(* Logix 5000 project; controller Prueba_Sintonizacion vendor 1 type 14 code 54 rev 20.15; software revision 20.04 *)

TASK MainTask (continuous, watchdog 500 ms) : MainProgram

MODULES
   Local : vendor 1 type 14 code 54 (ICP 0, rev 20.15)
END_MODULES

PROGRAM MainProgram   (* main routine MainRoutine *)
VAR
   Bit_prueba : BOOL;
   FCV_Flujo : REAL;
   PID : PID := (CTL := 8388608, PE := 1, SP := 30.0, KP := 0.029, KI := 61.247, KD := 15.352, MAXS := 100.0, MAXO := 100.0, UPD := 1.0, MAXI := 100.0, MAXCV := 100.0);
   PV_Temperature : REAL;
END_VAR

ROUTINE MainRoutine   (* ladder *)
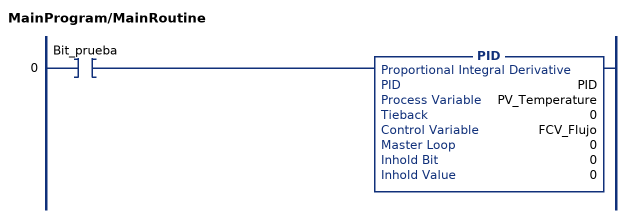
   0: XIC(Bit_prueba)PID(PID,PV_Temperature,0,FCV_Flujo,0,0,0);
END_ROUTINE
END_PROGRAM
